{attribute 'linkalways'} 
{attribute 'no_explicit_call' := 'This FB is a CLASS and must be accessed using methods or properties'}
{attribute 'enable_dynamic_creation'}
FUNCTION_BLOCK _ETcVnInterpolationType EXTENDS EnumDatatypeBase
VAR
	localData : ETcVnInterpolationType;
	activeData : REFERENCE TO ETcVnInterpolationType;
	enumBaseDatatype : _DINT(localData);
END_VAR

METHOD PRIVATE AddLocalEnumeration
VAR_INPUT
	Enumeration : T_MAXSTRING;
	Value : ETcVnInterpolationType;
END_VAR
AddEnumeration(Enumeration, Value);
END_METHOD

PROPERTY PUBLIC Address : PVOID
GET
Address := ADR(activeData);
END_GET
END_PROPERTY

METHOD PUBLIC ClearReference
VAR_INPUT
END_VAR
activeData REF= localData;
SetBaseDatatypeReference();
END_METHOD

METHOD PUBLIC Clone : I_Datatype
VAR
    pClone : POINTER TO _ETcVnInterpolationType;
END_VAR
pClone := __NEW(_ETcVnInterpolationType(InitialValue := Value));
Clone := pClone^;
END_METHOD

METHOD FB_init : BOOL
VAR_INPUT
	bInitRetains : BOOL; // if TRUE, the retain variables are initialized (warm start / cold start)
	bInCopyCode : BOOL;  // if TRUE, the instance afterwards gets moved into the copy code (online change)
	InitialValue : ETcVnInterpolationType;
END_VAR
localData := InitialValue;
AddBaseDatatype(enumBaseDatatype);
ClearReference();

AddLocalEnumeration('TCVN_IT_NEAREST_NEIGHBOR', ETcVnInterpolationType.TCVN_IT_NEAREST_NEIGHBOR);
AddLocalEnumeration('TCVN_IT_BILINEAR', ETcVnInterpolationType.TCVN_IT_BILINEAR);
AddLocalEnumeration('TCVN_IT_BICUBIC', ETcVnInterpolationType.TCVN_IT_BICUBIC);
AddLocalEnumeration('TCVN_IT_AREA_BASED', ETcVnInterpolationType.TCVN_IT_AREA_BASED);
AddLocalEnumeration('TCVN_IT_LANCZOS4', ETcVnInterpolationType.TCVN_IT_LANCZOS4);
END_METHOD

PROPERTY PUBLIC Identifier : T_MAXSTRING
GET
Identifier := 'ETcVnInterpolationType';
END_GET
END_PROPERTY

METHOD IsEnumeratorValueEqual : BOOL
VAR_INPUT
	Enumerator : I_KeyValueForwardEnumerator;
END_VAR
VAR
	storedValue : ETcVnInterpolationType;
END_VAR
IF NOT Enumerator.TryGet(storedValue) THEN
	RETURN;
END_IF

IsEnumeratorValueEqual := storedValue = activeData;
END_METHOD

METHOD PUBLIC MakeReferenceTo
VAR_INPUT
	ReferenceTarget : REFERENCE TO ETcVnInterpolationType;
END_VAR
activeData REF= ReferenceTarget;
SetBaseDatatypeReference();
END_METHOD

METHOD PROTECTED SetBaseDatatypeReference
VAR_INPUT
END_VAR
enumBaseDatatype.MakeReferenceTo(activeData);
END_METHOD

PROPERTY PUBLIC Size : UDINT
GET
Size := SIZEOF(activeData);
END_GET
END_PROPERTY

METHOD TryMakeReferenceTo : BOOL
VAR_INPUT
	Target : I_Datatype;
END_VAR
VAR
	targetAsEnum : I_EnumDatatype;
	pTargetData : POINTER TO ETcVnInterpolationType;
END_VAR
IF NOT Target.TryResolveAsEnumDatatype(targetAsEnum) THEN
	RETURN;
END_IF

IF targetAsEnum.Identifier <> Identifier THEN
	RETURN;
END_IF

pTargetData := Target.Address;
activeData REF= pTargetData^;
SetBaseDatatypeReference();
TryMakeReferenceTo := TRUE;
END_METHOD

PROPERTY PUBLIC Value : ETcVnInterpolationType
GET
Value := activeData;
END_GET
SET
activeData := Value;
END_SET
END_PROPERTY

END_FUNCTION_BLOCK

(* stored: Version 1.1.0.1, ProductVersion 3.1.4024.12
   POU _ETcVnInterpolationType: Id {20954bc4-43d2-40d0-94ee-ef3b742770fe}, SpecialFunc None
   Folder Constructor: Id {38f42632-f411-4f13-8358-e4eaae3cadc8}
   Folder Private: Id {0c14491a-5c3e-42db-8352-35890e0e59d9}
   Folder Protected: Id {254c20ee-63dc-4c6e-b220-7191b6c9bc9f}
   Method AddLocalEnumeration: Id {5f279f2c-beea-4cd3-a8dd-1cfefea61c07}
   Property Address: Id {e8b721c3-4bf2-4448-8862-b0248eca8e54}
   Get Get: Id {4dff995a-916a-4c8a-bae9-22c22a3bd554}
   Method ClearReference: Id {ad4ca338-7163-4877-8651-7611db3ad290}
   Method Clone: Id {a6638b55-e358-43ed-ba64-d7cd0af5a629}
   Method FB_init: Id {0aedc2f5-3a5c-4d2e-8266-563442b79577}
   Property Identifier: Id {58a7071a-f485-4a36-ae7a-f69342461031}
   Get Get: Id {a3b88427-cc87-43cf-b2dd-0de2ad23657f}
   Method IsEnumeratorValueEqual: Id {83da41cc-2a72-4563-8397-a4189a0b5c02}
   Method MakeReferenceTo: Id {c032b942-d633-436a-b09f-0067d2e0aaab}
   Method SetBaseDatatypeReference: Id {7df0615e-df9a-4add-a0be-27ba8429eaf8}
   Property Size: Id {6520a09c-4007-418c-9b7d-2c967f846df7}
   Get Get: Id {d6a9cdbf-a5a1-402a-95d8-86dc5d7f93eb}
   Method TryMakeReferenceTo: Id {9a7b9f69-d996-4a3d-87f1-eaaaf5519f61}
   Property Value: Id {fc2152ce-38e7-4567-91c4-19c3e44cc556}
   Get Get: Id {88170f08-7402-49db-b514-091a9c7eb799}
   Set Set: Id {254e05f0-a0b4-4934-8caf-17692219e033} *)
